TYPE ParameterSet :
STRUCT
	command : eCommandTypes := eCommandTypes.POSITION;
	parameter : ParameterGeneric;
END_STRUCT
END_TYPE

(* stored: Version 1.1.0.1, ProductVersion 3.1.4022.10
   DUT ParameterSet: Id {7787d46e-2a5f-4431-8438-c57dc843a3f1} *)
